FUNCTION_BLOCK Channel IMPLEMENTS I_Voltage
VAR_INPUT
END_VAR
VAR_OUTPUT
END_VAR
VAR
    _terminalAddress : WORD;
    _channelNumber : WORD;
    _guid : ChannelGuid;
    _name : STRING;
END_VAR

METHOD FB_init : BOOL
VAR_INPUT
	bInitRetains : BOOL; // if TRUE, the retain variables are initialized (warm start / cold start)
	bInCopyCode : BOOL;  // if TRUE, the instance afterwards gets moved into the copy code (online change)
    termianlAddress : WORD;
    channelNumber : WORD;
END_VAR
_terminalAddress := termianlAddress;
_channelNumber := channelNumber;
_guid.GuidCombo.ChannelNumber := _channelNumber;
_guid.GuidCombo.TerminalAddress := _terminalAddress;
END_METHOD

PROPERTY GUID : DWORD
GET
GUID := _guid.GuidValue;
END_GET
END_PROPERTY

PROPERTY Name : STRING
GET
Name := _name;
END_GET
SET
_name := Name;
END_SET
END_PROPERTY

END_FUNCTION_BLOCK

(* stored: Version 1.1.0.1, ProductVersion 3.1.4024.12
   POU Channel: Id {9f22b7fd-ffaa-470a-b4df-d8cbda897ecd}, SpecialFunc None
   Method FB_init: Id {582ecc2d-ba1b-4ba3-abf2-cdff45a9545b}
   Property GUID: Id {8fabec7f-c715-480e-a637-568fd5b5e6a0}
   Get Get: Id {7ddd41b5-6166-4fb6-8517-66e11cc7dfce}
   Property Name: Id {10914994-d070-4496-9266-05eef404ab11}
   Get Get: Id {96afc15d-73a9-4e78-8bbc-bc8bbc64d125}
   Set Set: Id {2e2289d7-a57b-4042-bea8-6bfd478489cd} *)
